FUNCTION_BLOCK FB_MeasurementStarted
VAR
	
	MeasurementValuesBuffer : ARRAY[1..gvl.MaxLoadMeasurementBufferSize] OF BYTE; 
	CurrentBufferIndiex : INT := 0;
	fbBuffer : FB_MemRingBuffer; 
	
	bReset : BOOL := TRUE; 
	bAdd : BOOL := TRUE;
	bGet : BOOL := TRUE;
	bRemove : BOOL := TRUE;
END_VAR

END_FUNCTION_BLOCK

(* stored: Version 1.1.0.1, ProductVersion 3.1.4024.12
   POU FB_MeasurementStarted: Id {86073582-c3eb-4a14-b9ea-908683465e53}, SpecialFunc None *)
